ABB RobotStudio station: Project1.rsstnx

Station Project1 (saved by RobotStudio 24.3.10958.1)
Controller Controller1, task T_ROB1: task frame (RAPID world) sits at (0, 0, 500) mm in the station
Controller Controller1
  mechanical unit ROB_1: IRB660_180_315__01, 6 joints, base frame (0, 0, 0) mm
Layout (positions relative to the parent item):
  - IRB660_180_315__01 [mechanism, from %ABB.RobotStudio.Models.IRB660%\IRB660_180_315__01.rslib] at (0, 0, 500) mm; joint values [-0.0436, 0.6621, 0.6612, -0.0431] (rad or m)
  - SC_PM_PLC [smart component, from Components\SC_PM_PLC.rslib]
      properties: SimulationQuickStart=All; StatisticsInfo=; con0_ID={00f7108f-041a-4658-8432-4663a157ed6e}; con0_pmPLC_dpSelectedFlowID=7507beaf-a637-4325-82e6-8dabecadb5e7; con0_T_ROB1_ID={ede59ae2-37f1-49be-aecb-80bcdd7f86de}; con0_T_ROB1_ObjectReleased=(none); pf1_Product_ToPick={da9875e8-a75e-44a1-b53a-961bb916f098}; pf1_PreparationTime_ToPick=1; pf1_Product_Placed=; pf1_ClearTime_Placed=0; pf1_ID=4b299c2b-0326-42f9-880b-26203f6d833c; pf2_Product_ToPick=; pf2_PreparationTime_ToPick=0; pf2_Product_Placed={660944ae-43fb-4d62-84a1-2b4997365d4d}; pf2_ClearTime_Placed=1; pf2_ID=081b0045-7d90-402c-a41a-05ee4f4aed6a; pf3_Product_ToPick={55fdd2c5-2514-4d7a-936c-0e237c314134}; pf3_PreparationTime_ToPick=1; pf3_Product_Placed=; pf3_ClearTime_Placed=0; pf3_ID=f450dbdc-584e-4e57-b0ab-3fff9d44f94b
  - Part_1 [part] at (-700, -600, 0) mm, size 1200 x 1200 x 500 mm
  - FlexGripper 2.0_Vacuum_Pallet [smart component, from Grippers\FlexGripper 2.0_Vacuum_Pallet.rslib] at (2410.12, -105.03, 1233.55) mm, rotated rx 180 ry 0 rz 179.98 deg
      properties: ReleasedObject=(none)
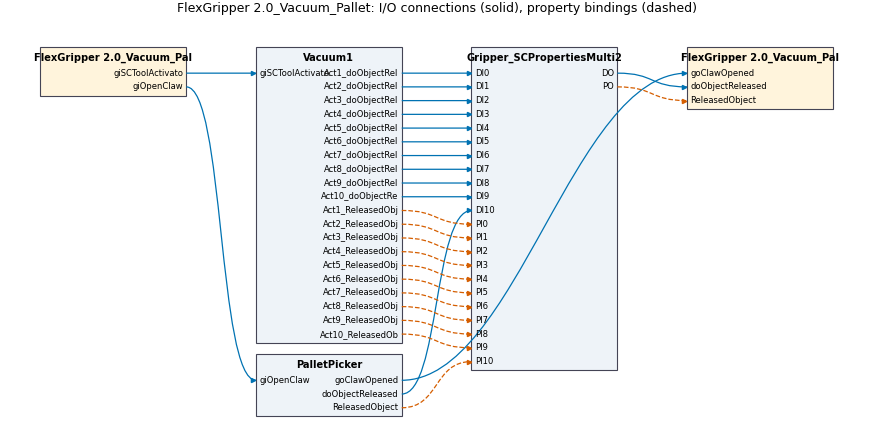
      connections:
        FlexGripper 2.0_Vacuum_Pallet.giSCToolActivators -> Vacuum1.giSCToolActivators
        FlexGripper 2.0_Vacuum_Pallet.giOpenClaw -> PalletPicker.giOpenClaw
        PalletPicker.goClawOpened -> FlexGripper 2.0_Vacuum_Pallet.goClawOpened
        Vacuum1.Act1_doObjectReleased -> Gripper_SCPropertiesMulti2Single.DI0
        Vacuum1.Act2_doObjectReleased -> Gripper_SCPropertiesMulti2Single.DI1
        Vacuum1.Act3_doObjectReleased -> Gripper_SCPropertiesMulti2Single.DI2
        Vacuum1.Act4_doObjectReleased -> Gripper_SCPropertiesMulti2Single.DI3
        Vacuum1.Act5_doObjectReleased -> Gripper_SCPropertiesMulti2Single.DI4
        Vacuum1.Act6_doObjectReleased -> Gripper_SCPropertiesMulti2Single.DI5
        Vacuum1.Act7_doObjectReleased -> Gripper_SCPropertiesMulti2Single.DI6
        Vacuum1.Act8_doObjectReleased -> Gripper_SCPropertiesMulti2Single.DI7
        Vacuum1.Act9_doObjectReleased -> Gripper_SCPropertiesMulti2Single.DI8
        Vacuum1.Act10_doObjectReleased -> Gripper_SCPropertiesMulti2Single.DI9
        PalletPicker.doObjectReleased -> Gripper_SCPropertiesMulti2Single.DI10
        Gripper_SCPropertiesMulti2Single.DO -> FlexGripper 2.0_Vacuum_Pallet.doObjectReleased
        Vacuum1.Act1_ReleasedObject => Gripper_SCPropertiesMulti2Single.PI0
        Vacuum1.Act2_ReleasedObject => Gripper_SCPropertiesMulti2Single.PI1
        Vacuum1.Act3_ReleasedObject => Gripper_SCPropertiesMulti2Single.PI2
        Vacuum1.Act4_ReleasedObject => Gripper_SCPropertiesMulti2Single.PI3
        Vacuum1.Act5_ReleasedObject => Gripper_SCPropertiesMulti2Single.PI4
        Vacuum1.Act6_ReleasedObject => Gripper_SCPropertiesMulti2Single.PI5
        Vacuum1.Act7_ReleasedObject => Gripper_SCPropertiesMulti2Single.PI6
        Vacuum1.Act8_ReleasedObject => Gripper_SCPropertiesMulti2Single.PI7
        Vacuum1.Act9_ReleasedObject => Gripper_SCPropertiesMulti2Single.PI8
        Vacuum1.Act10_ReleasedObject => Gripper_SCPropertiesMulti2Single.PI9
        PalletPicker.ReleasedObject => Gripper_SCPropertiesMulti2Single.PI10
        Gripper_SCPropertiesMulti2Single.PO => FlexGripper 2.0_Vacuum_Pallet.ReleasedObject
    - FlexGripper 2.0_Vacuum_Pallet [mechanism] at (0, 0, 0) mm; joint values [0, 0] (rad or m)
        TCP tVacuum at (0.12, 0.03, 163.81) mm, rotated rx 0 ry 0 rz -0.02 deg
        TCP tPalletPicker at (0.12, 0.03, 230.11) mm, rotated rx 0 ry 0 rz -0.02 deg
        links: L1, L2, L3, L4, L5, L6, L7
    - Vacuum1 [smart component]
        properties: Act1_ReleasedObject=(none); Act2_ReleasedObject=(none); Act3_ReleasedObject=(none); Act4_ReleasedObject=(none); Act5_ReleasedObject=(none); Act6_ReleasedObject=(none); Act7_ReleasedObject=(none); Act8_ReleasedObject=(none); Act9_ReleasedObject=(none); Act10_ReleasedObject=(none)
        signals: DO Act1_doObjectReleased, DO Act2_doObjectReleased, DO Act3_doObjectReleased, DO Act4_doObjectReleased, DO Act5_doObjectReleased, DO Act6_doObjectReleased, DO Act7_doObjectReleased, DO Act8_doObjectReleased, DO Act9_doObjectReleased, DO Act10_doObjectReleased, GI giSCToolActivators
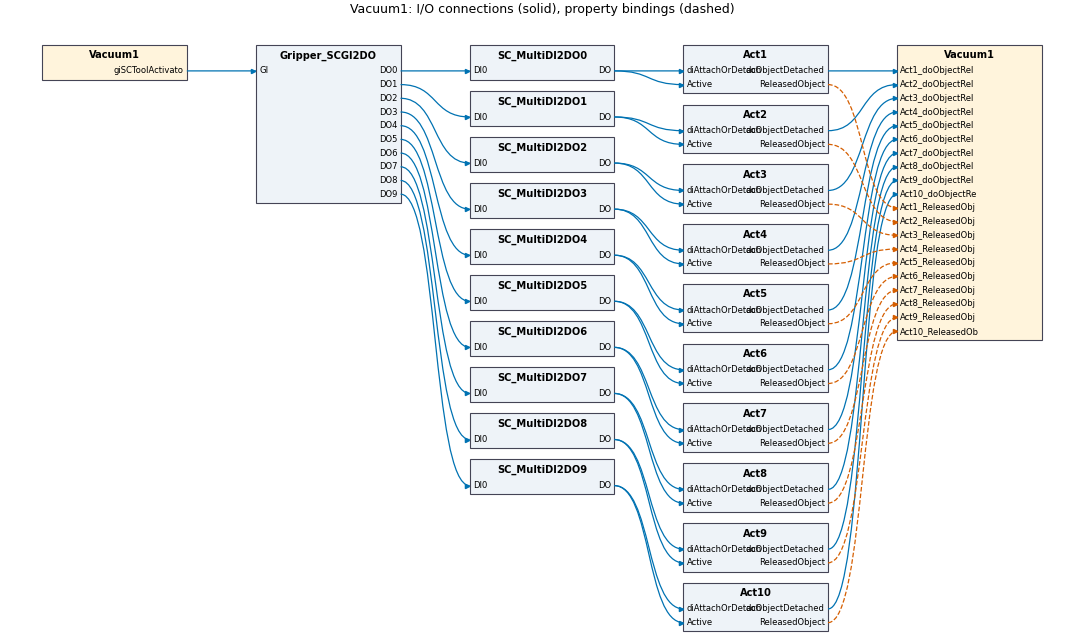
        connections:
          Act1.doObjectDetached -> Vacuum1.Act1_doObjectReleased
          Act2.doObjectDetached -> Vacuum1.Act2_doObjectReleased
          Act3.doObjectDetached -> Vacuum1.Act3_doObjectReleased
          Act4.doObjectDetached -> Vacuum1.Act4_doObjectReleased
          Act5.doObjectDetached -> Vacuum1.Act5_doObjectReleased
          Act6.doObjectDetached -> Vacuum1.Act6_doObjectReleased
          Act7.doObjectDetached -> Vacuum1.Act7_doObjectReleased
          Act8.doObjectDetached -> Vacuum1.Act8_doObjectReleased
          Act9.doObjectDetached -> Vacuum1.Act9_doObjectReleased
          Act10.doObjectDetached -> Vacuum1.Act10_doObjectReleased
          Gripper_SCGI2DO.DO0 -> SC_MultiDI2DO0.DI0
          SC_MultiDI2DO0.DO -> Act1.diAttachOrDetach
          SC_MultiDI2DO0.DO -> Act1.Active
          Gripper_SCGI2DO.DO1 -> SC_MultiDI2DO1.DI0
          SC_MultiDI2DO1.DO -> Act2.diAttachOrDetach
          SC_MultiDI2DO1.DO -> Act2.Active
          Gripper_SCGI2DO.DO2 -> SC_MultiDI2DO2.DI0
          SC_MultiDI2DO2.DO -> Act3.diAttachOrDetach
          SC_MultiDI2DO2.DO -> Act3.Active
          Gripper_SCGI2DO.DO3 -> SC_MultiDI2DO3.DI0
          SC_MultiDI2DO3.DO -> Act4.diAttachOrDetach
          SC_MultiDI2DO3.DO -> Act4.Active
          Gripper_SCGI2DO.DO4 -> SC_MultiDI2DO4.DI0
          SC_MultiDI2DO4.DO -> Act5.diAttachOrDetach
          SC_MultiDI2DO4.DO -> Act5.Active
          Gripper_SCGI2DO.DO5 -> SC_MultiDI2DO5.DI0
          SC_MultiDI2DO5.DO -> Act6.diAttachOrDetach
          SC_MultiDI2DO5.DO -> Act6.Active
          Gripper_SCGI2DO.DO6 -> SC_MultiDI2DO6.DI0
          SC_MultiDI2DO6.DO -> Act7.diAttachOrDetach
          SC_MultiDI2DO6.DO -> Act7.Active
          Gripper_SCGI2DO.DO7 -> SC_MultiDI2DO7.DI0
          SC_MultiDI2DO7.DO -> Act8.diAttachOrDetach
          SC_MultiDI2DO7.DO -> Act8.Active
          Gripper_SCGI2DO.DO8 -> SC_MultiDI2DO8.DI0
          SC_MultiDI2DO8.DO -> Act9.diAttachOrDetach
          SC_MultiDI2DO8.DO -> Act9.Active
          Gripper_SCGI2DO.DO9 -> SC_MultiDI2DO9.DI0
          SC_MultiDI2DO9.DO -> Act10.diAttachOrDetach
          SC_MultiDI2DO9.DO -> Act10.Active
          Vacuum1.giSCToolActivators -> Gripper_SCGI2DO.GI
          Act1.ReleasedObject => Vacuum1.Act1_ReleasedObject
          Act2.ReleasedObject => Vacuum1.Act2_ReleasedObject
          Act3.ReleasedObject => Vacuum1.Act3_ReleasedObject
          Act4.ReleasedObject => Vacuum1.Act4_ReleasedObject
          Act5.ReleasedObject => Vacuum1.Act5_ReleasedObject
          Act6.ReleasedObject => Vacuum1.Act6_ReleasedObject
          Act7.ReleasedObject => Vacuum1.Act7_ReleasedObject
          Act8.ReleasedObject => Vacuum1.Act8_ReleasedObject
          Act9.ReleasedObject => Vacuum1.Act9_ReleasedObject
          Act10.ReleasedObject => Vacuum1.Act10_ReleasedObject
      - Act1 [smart component] at (-0.1, -539.97, 163.81) mm, rotated rx 0 ry 0 rz -0.02 deg
          properties: ReleasedObject=(none); AttachedObject=(none)
          signals: DI diAttachOrDetach, DI Active, DO doObjectAttached, DO doObjectDetached
          connections:
            Act1.diAttachOrDetach -> SC_VolumeGripper.AttachOrDetach
            SC_VolumeGripper.TriggerAttach -> Attacher.Execute
            SC_VolumeGripper.TriggerDetach -> Detacher.Execute
            Attacher.Executed -> Act1.doObjectAttached
            Detacher.Executed -> Act1.doObjectDetached
            Act1.Active -> SC_VolumeGripper.Active
            SC_VolumeGripper.AttachParent => Attacher.Parent
            SC_VolumeGripper.ChildToAttach => Attacher.Child
            SC_VolumeGripper.AttachedChild => Detacher.Child
            SC_VolumeGripper.AttachedChild => Act1.AttachedObject
            SC_VolumeGripper.ReleasedChild => Act1.ReleasedObject
        - SC_VolumeGripper [smart component, from Components\SC_VolumeGripper.rslib]
            properties: Position=[0 0 0]; Orientation=[0 0 0]; Size=[0.28 0.1 0.02]; AttachParent=Act1; ChildToAttach=(none); AttachedChild=(none); ReleasedChild=(none)
          - _sensorPart_ [part], size 280 x 100 x 20 mm
        - Attacher [smart component, from Components\Attacher.rslib]
            properties: Parent=Act1; Flange=0; Child=(none); Mount=false; Offset=[0 0 0]; Orientation=[0 0 0]
        - Detacher [smart component, from Components\Detacher.rslib]
            properties: Child=(none); KeepPosition=true
      - Act2 [smart component] at (-0.05, -419.97, 163.81) mm, rotated rx 0 ry 0 rz -0.02 deg
          properties: ReleasedObject=(none); AttachedObject=(none)
          signals: DI diAttachOrDetach, DI Active, DO doObjectAttached, DO doObjectDetached
          connections:
            Act2.diAttachOrDetach -> SC_VolumeGripper.AttachOrDetach
            SC_VolumeGripper.TriggerAttach -> Attacher.Execute
            SC_VolumeGripper.TriggerDetach -> Detacher.Execute
            Attacher.Executed -> Act2.doObjectAttached
            Detacher.Executed -> Act2.doObjectDetached
            Act2.Active -> SC_VolumeGripper.Active
            SC_VolumeGripper.AttachParent => Attacher.Parent
            SC_VolumeGripper.ChildToAttach => Attacher.Child
            SC_VolumeGripper.AttachedChild => Detacher.Child
            SC_VolumeGripper.AttachedChild => Act2.AttachedObject
            SC_VolumeGripper.ReleasedChild => Act2.ReleasedObject
        - SC_VolumeGripper [smart component, from Components\SC_VolumeGripper.rslib]
            properties: Position=[0 0 0]; Orientation=[0 0 0]; Size=[0.28 0.1 0.02]; AttachParent=Act2; ChildToAttach=(none); AttachedChild=(none); ReleasedChild=(none)
          - _sensorPart_ [part], size 280 x 100 x 20 mm
        - Attacher [smart component, from Components\Attacher.rslib]
            properties: Parent=Act2; Flange=0; Child=(none); Mount=false; Offset=[0 0 0]; Orientation=[0 0 0]
        - Detacher [smart component, from Components\Detacher.rslib]
            properties: Child=(none); KeepPosition=true
      - Act3 [smart component] at (0, -299.97, 163.81) mm, rotated rx 0 ry 0 rz -0.02 deg
          properties: ReleasedObject=(none); AttachedObject=(none)
          signals: DI diAttachOrDetach, DI Active, DO doObjectAttached, DO doObjectDetached
          connections:
            Act3.diAttachOrDetach -> SC_VolumeGripper.AttachOrDetach
            SC_VolumeGripper.TriggerAttach -> Attacher.Execute
            SC_VolumeGripper.TriggerDetach -> Detacher.Execute
            Attacher.Executed -> Act3.doObjectAttached
            Detacher.Executed -> Act3.doObjectDetached
            Act3.Active -> SC_VolumeGripper.Active
            SC_VolumeGripper.AttachParent => Attacher.Parent
            SC_VolumeGripper.ChildToAttach => Attacher.Child
            SC_VolumeGripper.AttachedChild => Detacher.Child
            SC_VolumeGripper.AttachedChild => Act3.AttachedObject
            SC_VolumeGripper.ReleasedChild => Act3.ReleasedObject
        - SC_VolumeGripper [smart component, from Components\SC_VolumeGripper.rslib]
            properties: Position=[0 0 0]; Orientation=[0 0 0]; Size=[0.28 0.1 0.02]; AttachParent=Act3; ChildToAttach=(none); AttachedChild=(none); ReleasedChild=(none)
          - _sensorPart_ [part], size 280 x 100 x 20 mm
        - Attacher [smart component, from Components\Attacher.rslib]
            properties: Parent=Act3; Flange=0; Child=(none); Mount=false; Offset=[0 0 0]; Orientation=[0 0 0]
        - Detacher [smart component, from Components\Detacher.rslib]
            properties: Child=(none); KeepPosition=true
      - Act4 [smart component] at (0.05, -179.97, 163.81) mm, rotated rx 0 ry 0 rz -0.02 deg
          properties: ReleasedObject=(none); AttachedObject=(none)
          signals: DI diAttachOrDetach, DI Active, DO doObjectAttached, DO doObjectDetached
          connections:
            Act4.diAttachOrDetach -> SC_VolumeGripper.AttachOrDetach
            SC_VolumeGripper.TriggerAttach -> Attacher.Execute
            SC_VolumeGripper.TriggerDetach -> Detacher.Execute
            Attacher.Executed -> Act4.doObjectAttached
            Detacher.Executed -> Act4.doObjectDetached
            Act4.Active -> SC_VolumeGripper.Active
            SC_VolumeGripper.AttachParent => Attacher.Parent
            SC_VolumeGripper.ChildToAttach => Attacher.Child
            SC_VolumeGripper.AttachedChild => Detacher.Child
            SC_VolumeGripper.AttachedChild => Act4.AttachedObject
            SC_VolumeGripper.ReleasedChild => Act4.ReleasedObject
        - SC_VolumeGripper [smart component, from Components\SC_VolumeGripper.rslib]
            properties: Position=[0 0 0]; Orientation=[0 0 0]; Size=[0.28 0.1 0.02]; AttachParent=Act4; ChildToAttach=(none); AttachedChild=(none); ReleasedChild=(none)
          - _sensorPart_ [part], size 280 x 100 x 20 mm
        - Attacher [smart component, from Components\Attacher.rslib]
            properties: Parent=Act4; Flange=0; Child=(none); Mount=false; Offset=[0 0 0]; Orientation=[0 0 0]
        - Detacher [smart component, from Components\Detacher.rslib]
            properties: Child=(none); KeepPosition=true
      - Act5 [smart component] at (0.1, -59.97, 163.81) mm, rotated rx 0 ry 0 rz -0.02 deg
          properties: ReleasedObject=(none); AttachedObject=(none)
          signals: DI diAttachOrDetach, DI Active, DO doObjectAttached, DO doObjectDetached
          connections:
            Act5.diAttachOrDetach -> SC_VolumeGripper.AttachOrDetach
            SC_VolumeGripper.TriggerAttach -> Attacher.Execute
            SC_VolumeGripper.TriggerDetach -> Detacher.Execute
            Attacher.Executed -> Act5.doObjectAttached
            Detacher.Executed -> Act5.doObjectDetached
            Act5.Active -> SC_VolumeGripper.Active
            SC_VolumeGripper.AttachParent => Attacher.Parent
            SC_VolumeGripper.ChildToAttach => Attacher.Child
            SC_VolumeGripper.AttachedChild => Detacher.Child
            SC_VolumeGripper.AttachedChild => Act5.AttachedObject
            SC_VolumeGripper.ReleasedChild => Act5.ReleasedObject
        - SC_VolumeGripper [smart component, from Components\SC_VolumeGripper.rslib]
            properties: Position=[0 0 0]; Orientation=[0 0 0]; Size=[0.28 0.1 0.02]; AttachParent=Act5; ChildToAttach=(none); AttachedChild=(none); ReleasedChild=(none)
          - _sensorPart_ [part], size 280 x 100 x 20 mm
        - Attacher [smart component, from Components\Attacher.rslib]
            properties: Parent=Act5; Flange=0; Child=(none); Mount=false; Offset=[0 0 0]; Orientation=[0 0 0]
        - Detacher [smart component, from Components\Detacher.rslib]
            properties: Child=(none); KeepPosition=true
      - Act6 [smart component] at (0.14, 60.03, 163.81) mm, rotated rx 0 ry 0 rz -0.02 deg
          properties: ReleasedObject=(none); AttachedObject=(none)
          signals: DI diAttachOrDetach, DI Active, DO doObjectAttached, DO doObjectDetached
          connections:
            Act6.diAttachOrDetach -> SC_VolumeGripper.AttachOrDetach
            SC_VolumeGripper.TriggerAttach -> Attacher.Execute
            SC_VolumeGripper.TriggerDetach -> Detacher.Execute
            Attacher.Executed -> Act6.doObjectAttached
            Detacher.Executed -> Act6.doObjectDetached
            Act6.Active -> SC_VolumeGripper.Active
            SC_VolumeGripper.AttachParent => Attacher.Parent
            SC_VolumeGripper.ChildToAttach => Attacher.Child
            SC_VolumeGripper.AttachedChild => Detacher.Child
            SC_VolumeGripper.AttachedChild => Act6.AttachedObject
            SC_VolumeGripper.ReleasedChild => Act6.ReleasedObject
        - SC_VolumeGripper [smart component, from Components\SC_VolumeGripper.rslib]
            properties: Position=[0 0 0]; Orientation=[0 0 0]; Size=[0.28 0.1 0.02]; AttachParent=Act6; ChildToAttach=(none); AttachedChild=(none); ReleasedChild=(none)
          - _sensorPart_ [part], size 280 x 100 x 20 mm
        - Attacher [smart component, from Components\Attacher.rslib]
            properties: Parent=Act6; Flange=0; Child=(none); Mount=false; Offset=[0 0 0]; Orientation=[0 0 0]
        - Detacher [smart component, from Components\Detacher.rslib]
            properties: Child=(none); KeepPosition=true
      - Act7 [smart component] at (0.19, 180.03, 163.81) mm, rotated rx 0 ry 0 rz -0.02 deg
          properties: ReleasedObject=(none); AttachedObject=(none)
          signals: DI diAttachOrDetach, DI Active, DO doObjectAttached, DO doObjectDetached
          connections:
            Act7.diAttachOrDetach -> SC_VolumeGripper.AttachOrDetach
            SC_VolumeGripper.TriggerAttach -> Attacher.Execute
            SC_VolumeGripper.TriggerDetach -> Detacher.Execute
            Attacher.Executed -> Act7.doObjectAttached
            Detacher.Executed -> Act7.doObjectDetached
            Act7.Active -> SC_VolumeGripper.Active
            SC_VolumeGripper.AttachParent => Attacher.Parent
            SC_VolumeGripper.ChildToAttach => Attacher.Child
            SC_VolumeGripper.AttachedChild => Detacher.Child
            SC_VolumeGripper.AttachedChild => Act7.AttachedObject
            SC_VolumeGripper.ReleasedChild => Act7.ReleasedObject
        - SC_VolumeGripper [smart component, from Components\SC_VolumeGripper.rslib]
            properties: Position=[0 0 0]; Orientation=[0 0 0]; Size=[0.28 0.1 0.02]; AttachParent=Act7; ChildToAttach=(none); AttachedChild=(none); ReleasedChild=(none)
          - _sensorPart_ [part], size 280 x 100 x 20 mm
        - Attacher [smart component, from Components\Attacher.rslib]
            properties: Parent=Act7; Flange=0; Child=(none); Mount=false; Offset=[0 0 0]; Orientation=[0 0 0]
        - Detacher [smart component, from Components\Detacher.rslib]
            properties: Child=(none); KeepPosition=true
      - Act8 [smart component] at (0.24, 300.03, 163.81) mm, rotated rx 0 ry 0 rz -0.02 deg
          properties: ReleasedObject=(none); AttachedObject=(none)
          signals: DI diAttachOrDetach, DI Active, DO doObjectAttached, DO doObjectDetached
          connections:
            Act8.diAttachOrDetach -> SC_VolumeGripper.AttachOrDetach
            SC_VolumeGripper.TriggerAttach -> Attacher.Execute
            SC_VolumeGripper.TriggerDetach -> Detacher.Execute
            Attacher.Executed -> Act8.doObjectAttached
            Detacher.Executed -> Act8.doObjectDetached
            Act8.Active -> SC_VolumeGripper.Active
            SC_VolumeGripper.AttachParent => Attacher.Parent
            SC_VolumeGripper.ChildToAttach => Attacher.Child
            SC_VolumeGripper.AttachedChild => Detacher.Child
            SC_VolumeGripper.AttachedChild => Act8.AttachedObject
            SC_VolumeGripper.ReleasedChild => Act8.ReleasedObject
        - SC_VolumeGripper [smart component, from Components\SC_VolumeGripper.rslib]
            properties: Position=[0 0 0]; Orientation=[0 0 0]; Size=[0.28 0.1 0.02]; AttachParent=Act8; ChildToAttach=(none); AttachedChild=(none); ReleasedChild=(none)
          - _sensorPart_ [part], size 280 x 100 x 20 mm
        - Attacher [smart component, from Components\Attacher.rslib]
            properties: Parent=Act8; Flange=0; Child=(none); Mount=false; Offset=[0 0 0]; Orientation=[0 0 0]
        - Detacher [smart component, from Components\Detacher.rslib]
            properties: Child=(none); KeepPosition=true
      - Act9 [smart component] at (0.29, 420.03, 163.81) mm, rotated rx 0 ry 0 rz -0.02 deg
          properties: ReleasedObject=(none); AttachedObject=(none)
          signals: DI diAttachOrDetach, DI Active, DO doObjectAttached, DO doObjectDetached
          connections:
            Act9.diAttachOrDetach -> SC_VolumeGripper.AttachOrDetach
            SC_VolumeGripper.TriggerAttach -> Attacher.Execute
            SC_VolumeGripper.TriggerDetach -> Detacher.Execute
            Attacher.Executed -> Act9.doObjectAttached
            Detacher.Executed -> Act9.doObjectDetached
            Act9.Active -> SC_VolumeGripper.Active
            SC_VolumeGripper.AttachParent => Attacher.Parent
            SC_VolumeGripper.ChildToAttach => Attacher.Child
            SC_VolumeGripper.AttachedChild => Detacher.Child
            SC_VolumeGripper.AttachedChild => Act9.AttachedObject
            SC_VolumeGripper.ReleasedChild => Act9.ReleasedObject
        - SC_VolumeGripper [smart component, from Components\SC_VolumeGripper.rslib]
            properties: Position=[0 0 0]; Orientation=[0 0 0]; Size=[0.28 0.1 0.02]; AttachParent=Act9; ChildToAttach=(none); AttachedChild=(none); ReleasedChild=(none)
          - _sensorPart_ [part], size 280 x 100 x 20 mm
        - Attacher [smart component, from Components\Attacher.rslib]
            properties: Parent=Act9; Flange=0; Child=(none); Mount=false; Offset=[0 0 0]; Orientation=[0 0 0]
        - Detacher [smart component, from Components\Detacher.rslib]
            properties: Child=(none); KeepPosition=true
      - Act10 [smart component] at (0.34, 540.03, 163.81) mm, rotated rx 0 ry 0 rz -0.02 deg
          properties: ReleasedObject=(none); AttachedObject=(none)
          signals: DI diAttachOrDetach, DI Active, DO doObjectAttached, DO doObjectDetached
          connections:
            Act10.diAttachOrDetach -> SC_VolumeGripper.AttachOrDetach
            SC_VolumeGripper.TriggerAttach -> Attacher.Execute
            SC_VolumeGripper.TriggerDetach -> Detacher.Execute
            Attacher.Executed -> Act10.doObjectAttached
            Detacher.Executed -> Act10.doObjectDetached
            Act10.Active -> SC_VolumeGripper.Active
            SC_VolumeGripper.AttachParent => Attacher.Parent
            SC_VolumeGripper.ChildToAttach => Attacher.Child
            SC_VolumeGripper.AttachedChild => Detacher.Child
            SC_VolumeGripper.AttachedChild => Act10.AttachedObject
            SC_VolumeGripper.ReleasedChild => Act10.ReleasedObject
        - SC_VolumeGripper [smart component, from Components\SC_VolumeGripper.rslib]
            properties: Position=[0 0 0]; Orientation=[0 0 0]; Size=[0.28 0.1 0.02]; AttachParent=Act10; ChildToAttach=(none); AttachedChild=(none); ReleasedChild=(none)
          - _sensorPart_ [part], size 280 x 100 x 20 mm
        - Attacher [smart component, from Components\Attacher.rslib]
            properties: Parent=Act10; Flange=0; Child=(none); Mount=false; Offset=[0 0 0]; Orientation=[0 0 0]
        - Detacher [smart component, from Components\Detacher.rslib]
            properties: Child=(none); KeepPosition=true
      - Gripper_SCGI2DO [smart component, from Components\SC_GI2DO.rslib]
          properties: DOCount=11
      - SC_MultiDI2DO0 [smart component, from Components\SC_MultiDI2DO.rslib]
          properties: DICount=1; ConnectionType=0/1
      - SC_MultiDI2DO1 [smart component, from Components\SC_MultiDI2DO.rslib]
          properties: DICount=1; ConnectionType=0/1
      - SC_MultiDI2DO2 [smart component, from Components\SC_MultiDI2DO.rslib]
          properties: DICount=1; ConnectionType=0/1
      - SC_MultiDI2DO3 [smart component, from Components\SC_MultiDI2DO.rslib]
          properties: DICount=1; ConnectionType=0/1
      - SC_MultiDI2DO4 [smart component, from Components\SC_MultiDI2DO.rslib]
          properties: DICount=1; ConnectionType=0/1
      - SC_MultiDI2DO5 [smart component, from Components\SC_MultiDI2DO.rslib]
          properties: DICount=1; ConnectionType=0/1
      - SC_MultiDI2DO6 [smart component, from Components\SC_MultiDI2DO.rslib]
          properties: DICount=1; ConnectionType=0/1
      - SC_MultiDI2DO7 [smart component, from Components\SC_MultiDI2DO.rslib]
          properties: DICount=1; ConnectionType=0/1
      - SC_MultiDI2DO8 [smart component, from Components\SC_MultiDI2DO.rslib]
          properties: DICount=1; ConnectionType=0/1
      - SC_MultiDI2DO9 [smart component, from Components\SC_MultiDI2DO.rslib]
          properties: DICount=1; ConnectionType=0/1
    - PalletPicker [smart component]
        properties: ReleasedObject=(none)
        signals: GI giOpenClaw, GO goClawOpened, DO doObjectReleased
        connections:
          PalletPicker.giOpenClaw -> ClawControl.giOpenClaw
          ClawControl.goClawOpened -> PalletPicker.goClawOpened
          ClawAct.doObjectDetached -> PalletPicker.doObjectReleased
          ClawControl.Closed -> LogicSRLatch.Set
          ClawControl.Opening -> LogicSRLatch.Reset
          LogicSRLatch.Output -> ClawAct.diAttachOrDetach
          ClawControl.Closed -> LogicGate.InputA
          ClawControl.Opening -> LogicGate.InputB
          LogicGate.Output -> ClawAct.Active
          ClawAct.ReleasedObject => PalletPicker.ReleasedObject
      - ClawControl [smart component]
          signals: GI giOpenClaw, GO goClawOpened, DO Closing, DO Closed, DO Opening, DO Opened
          connections:
            JointMoverClose.Executing -> ClawControl.Closing
            JointMoverClose.Executed -> ClawControl.Closed
            JointMoverOpen.Executing -> ClawControl.Opening
            JointMoverOpen.Executed -> ClawControl.Opened
            ClawControl.giOpenClaw -> MultiSignalJudgeOpen.GI0
            MultiSignalJudgeOpen.DO -> JointMoverOpen.Execute
            JointMoverOpen.Executed -> MultiSignalSetOpen.Set
            ClawControl.giOpenClaw -> MultiSignalJudgeClose.GI0
            MultiSignalJudgeClose.DO -> JointMoverClose.Execute
            JointMoverClose.Executed -> MultiSignalSetClose.Set
            MultiSignalSetOpen.Executed -> MutiSignalSelector.SelectorA
            MultiSignalSetOpen.GO0 -> MutiSignalSelector.GiA0
            MultiSignalSetClose.Executed -> MutiSignalSelector.SelectorB
            MultiSignalSetClose.GO0 -> MutiSignalSelector.GiB0
            MutiSignalSelector.goClawOpened -> ClawControl.goClawOpened
        - MultiSignalJudgeOpen [smart component, from Components\SC_MultiSignalJudge.rslib]
            properties: DICount=0; GICount=1
        - JointMoverOpen [smart component, from Components\SC_JointMoverEx.rslib]
            properties: Mechanism=FlexGripper 2.0_Vacuum_Pallet; Relative=false; Duration=0.5; UseJ1=true; J1=0.1; UseJ2=true; J2=0.1
        - MultiSignalSetOpen [smart component, from Components\SC_MultiSignalSet.rslib]
            properties: DOCount=0; GOCount=1
        - MultiSignalJudgeClose [smart component, from Components\SC_MultiSignalJudge.rslib]
            properties: DICount=0; GICount=1
        - JointMoverClose [smart component, from Components\SC_JointMoverEx.rslib]
            properties: Mechanism=FlexGripper 2.0_Vacuum_Pallet; Relative=false; Duration=0.5; UseJ1=true; J1=0; UseJ2=true; J2=0
        - MultiSignalSetClose [smart component, from Components\SC_MultiSignalSet.rslib]
            properties: DOCount=0; GOCount=1
        - MutiSignalSelector [smart component, from Components\SC_MultiSignalSelector.rslib]
            properties: DICountA=0; GICountA=1; DICountB=0; GICountB=1; PiGiA0=goClawOpened; PiGiB0=goClawOpened
      - ClawAct [smart component] at (0.12, 0.03, 180.11) mm, rotated rx 0 ry 0 rz -0.02 deg
          properties: ReleasedObject=(none); AttachedObject=(none)
          signals: DI diAttachOrDetach, DI Active, DO doObjectAttached, DO doObjectDetached
          connections:
            ClawAct.diAttachOrDetach -> SC_VolumeGripper.AttachOrDetach
            SC_VolumeGripper.TriggerAttach -> Attacher.Execute
            SC_VolumeGripper.TriggerDetach -> Detacher.Execute
            Attacher.Executed -> ClawAct.doObjectAttached
            Detacher.Executed -> ClawAct.doObjectDetached
            ClawAct.Active -> SC_VolumeGripper.Active
            SC_VolumeGripper.AttachParent => Attacher.Parent
            SC_VolumeGripper.ChildToAttach => Attacher.Child
            SC_VolumeGripper.AttachedChild => Detacher.Child
            SC_VolumeGripper.AttachedChild => ClawAct.AttachedObject
            SC_VolumeGripper.ReleasedChild => ClawAct.ReleasedObject
        - SC_VolumeGripper [smart component, from Components\SC_VolumeGripper.rslib]
            properties: Position=[0 0 0]; Orientation=[0 0 0]; Size=[0.02 1.2 0.08]; AttachParent=ClawAct; ChildToAttach=(none); AttachedChild=(none); ReleasedChild=(none)
          - _sensorPart_ [part], size 20 x 1200 x 80 mm
        - Attacher [smart component, from Components\Attacher.rslib]
            properties: Parent=ClawAct; Flange=0; Child=(none); Mount=false; Offset=[0 0 0]; Orientation=[0 0 0]
        - Detacher [smart component, from Components\Detacher.rslib]
            properties: Child=(none); KeepPosition=true
      - LogicSRLatch [smart component, from Components\LogicSRLatch.rslib]
      - LogicGate [smart component, from Components\LogicGate.rslib]
          properties: Operator=OR; Delay=0
    - Gripper_SCPropertiesMulti2Single [smart component, from Components\SC_PropertiesMulti2Single.rslib]
        properties: Count=11; PO=(none); PI0=(none); PI1=(none); PI2=(none); PI3=(none); PI4=(none); PI5=(none); PI6=(none); PI7=(none); PI8=(none); PI9=(none); PI10=(none)
  - Conveyor_600 [smart component, from Feeders\Conveyor_600.rslib] at (800, 2100, 0) mm, rotated rx 0 ry 0 rz 90 deg
      properties: PreparationTime_ToPick=1; Product_ToPick={da9875e8-a75e-44a1-b53a-961bb916f098}; ClearTime_Placed=0; Product_Placed=
      connections:
        Conveyor_600.Reset -> SCFeederController.Reset
        Conveyor_600.Enqueue_ToPick -> SCFeederController.Enqueue_ToPick
        SCFeederController.Shown_ToPick -> Conveyor_600.Shown_ToPick
        Conveyor_600.Clear_ToPick -> SCFeederController.Clear_ToPick
        Conveyor_600.GI_ProdSel_ToPick -> SCFeederController.GI_ProdSel_ToPick
        Conveyor_600.GI_FormSel_ToPick -> SCFeederController.GI_FormSel_ToPick
        SCFeederController.GO_ProdSel_ToPick -> Conveyor_600.GO_ProdSel_ToPick
        SCFeederController.GO_FormSel_ToPick -> Conveyor_600.GO_FormSel_ToPick
        SCFeederController.Clear_Placed_Finished -> Conveyor_600.Clear_Placed_Finished
        Conveyor_600.Enqueue_Placed -> SCFeederController.Enqueue_Placed
        Conveyor_600.Clear_Placed -> SCFeederController.Clear_Placed
        Conveyor_600.Enqueue_IOPlacedRequest -> SCFeederController.Enqueue_IOPlacedRequest
        Conveyor_600.GI_ProdSel_PlacedRequest -> SCFeederController.GI_ProdSel_PlacedRequest
        Conveyor_600.GI_FormSel_PlacedRequest -> SCFeederController.GI_FormSel_PlacedRequest
        SCFeederController.GO_ProdSel_PlacedRequest -> Conveyor_600.GO_ProdSel_PlacedRequest
        SCFeederController.GO_FormSel_PlacedRequest -> Conveyor_600.GO_FormSel_PlacedRequest
        SCFeederController.IsReady_IOPlacedRequest -> Conveyor_600.IsReady_IOPlacedRequest
        Conveyor_600.PreparationTime_ToPick => SCFeederController.PreparationTime_ToPick
        Conveyor_600.Product_ToPick => SCFeederController.Product_ToPick
        Conveyor_600.ClearTime_Placed => SCFeederController.ClearTime_Placed
        Conveyor_600.Product_Placed => SCFeederController.Product_Placed
    - 600_guide [part, from Feeders\Conveyor_600.rslib]
    - SCFeederController [smart component, from Components\SC_FeederController.rslib]
        properties: Product_Placed=; ClearTime_Placed=0; PreparationTime_ToPick=1; Product_ToPick={da9875e8-a75e-44a1-b53a-961bb916f098}
  - Outfeeder_1320 [smart component, from Feeders\Outfeeder_1320.rslib] at (1600, -700, 0) mm
      properties: PreparationTime_ToPick=0; Product_ToPick=; ClearTime_Placed=1; Product_Placed={660944ae-43fb-4d62-84a1-2b4997365d4d}
      connections:
        Outfeeder_1320.Reset -> SCFeederController.Reset
        Outfeeder_1320.Enqueue_ToPick -> SCFeederController.Enqueue_ToPick
        SCFeederController.Shown_ToPick -> Outfeeder_1320.Shown_ToPick
        Outfeeder_1320.Clear_ToPick -> SCFeederController.Clear_ToPick
        Outfeeder_1320.GI_ProdSel_ToPick -> SCFeederController.GI_ProdSel_ToPick
        Outfeeder_1320.GI_FormSel_ToPick -> SCFeederController.GI_FormSel_ToPick
        SCFeederController.GO_ProdSel_ToPick -> Outfeeder_1320.GO_ProdSel_ToPick
        SCFeederController.GO_FormSel_ToPick -> Outfeeder_1320.GO_FormSel_ToPick
        SCFeederController.Clear_Placed_Finished -> Outfeeder_1320.Clear_Placed_Finished
        Outfeeder_1320.Enqueue_Placed -> SCFeederController.Enqueue_Placed
        Outfeeder_1320.Clear_Placed -> SCFeederController.Clear_Placed
        Outfeeder_1320.Enqueue_IOPlacedRequest -> SCFeederController.Enqueue_IOPlacedRequest
        Outfeeder_1320.GI_ProdSel_PlacedRequest -> SCFeederController.GI_ProdSel_PlacedRequest
        Outfeeder_1320.GI_FormSel_PlacedRequest -> SCFeederController.GI_FormSel_PlacedRequest
        SCFeederController.GO_ProdSel_PlacedRequest -> Outfeeder_1320.GO_ProdSel_PlacedRequest
        SCFeederController.GO_FormSel_PlacedRequest -> Outfeeder_1320.GO_FormSel_PlacedRequest
        SCFeederController.IsReady_IOPlacedRequest -> Outfeeder_1320.IsReady_IOPlacedRequest
        Outfeeder_1320.PreparationTime_ToPick => SCFeederController.PreparationTime_ToPick
        Outfeeder_1320.Product_ToPick => SCFeederController.Product_ToPick
        Outfeeder_1320.ClearTime_Placed => SCFeederController.ClearTime_Placed
        Outfeeder_1320.Product_Placed => SCFeederController.Product_Placed
    - 1320_4000_h2 [part, from Feeders\Outfeeder_1320.rslib]
    - SCFeederController [smart component, from Components\SC_FeederController.rslib]
        properties: Product_Placed={660944ae-43fb-4d62-84a1-2b4997365d4d}; ClearTime_Placed=1; PreparationTime_ToPick=0; Product_ToPick=
  - PalletDispenser 1300_1300_300 [smart component, from Feeders\PalletDispenser 1300_1300_300.rslib] at (-300, -1600, 0) mm, rotated rx 0 ry 0 rz -90 deg
      properties: PreparationTime_ToPick=1; Product_ToPick={55fdd2c5-2514-4d7a-936c-0e237c314134}; ClearTime_Placed=0; Product_Placed=
      connections:
        PalletDispenser 1300_1300_300.Reset -> SCFeederController.Reset
        PalletDispenser 1300_1300_300.Enqueue_ToPick -> SCFeederController.Enqueue_ToPick
        SCFeederController.Shown_ToPick -> PalletDispenser 1300_1300_300.Shown_ToPick
        PalletDispenser 1300_1300_300.Clear_ToPick -> SCFeederController.Clear_ToPick
        PalletDispenser 1300_1300_300.GI_ProdSel_ToPick -> SCFeederController.GI_ProdSel_ToPick
        PalletDispenser 1300_1300_300.GI_FormSel_ToPick -> SCFeederController.GI_FormSel_ToPick
        SCFeederController.GO_ProdSel_ToPick -> PalletDispenser 1300_1300_300.GO_ProdSel_ToPick
        SCFeederController.GO_FormSel_ToPick -> PalletDispenser 1300_1300_300.GO_FormSel_ToPick
        SCFeederController.Clear_Placed_Finished -> PalletDispenser 1300_1300_300.Clear_Placed_Finished
        PalletDispenser 1300_1300_300.Enqueue_Placed -> SCFeederController.Enqueue_Placed
        PalletDispenser 1300_1300_300.Clear_Placed -> SCFeederController.Clear_Placed
        PalletDispenser 1300_1300_300.Enqueue_IOPlacedRequest -> SCFeederController.Enqueue_IOPlacedRequest
        PalletDispenser 1300_1300_300.GI_ProdSel_PlacedRequest -> SCFeederController.GI_ProdSel_PlacedRequest
        PalletDispenser 1300_1300_300.GI_FormSel_PlacedRequest -> SCFeederController.GI_FormSel_PlacedRequest
        SCFeederController.GO_ProdSel_PlacedRequest -> PalletDispenser 1300_1300_300.GO_ProdSel_PlacedRequest
        SCFeederController.GO_FormSel_PlacedRequest -> PalletDispenser 1300_1300_300.GO_FormSel_PlacedRequest
        SCFeederController.IsReady_IOPlacedRequest -> PalletDispenser 1300_1300_300.IsReady_IOPlacedRequest
        PalletDispenser 1300_1300_300.PreparationTime_ToPick => SCFeederController.PreparationTime_ToPick
        PalletDispenser 1300_1300_300.Product_ToPick => SCFeederController.Product_ToPick
        PalletDispenser 1300_1300_300.ClearTime_Placed => SCFeederController.ClearTime_Placed
        PalletDispenser 1300_1300_300.Product_Placed => SCFeederController.Product_Placed
    - PalletDispenser 1300_1300_300 [part, from Feeders\PalletDispenser 1300_1300_300.rslib]
    - SCFeederController [smart component, from Components\SC_FeederController.rslib]
        properties: Product_Placed=; ClearTime_Placed=0; PreparationTime_ToPick=1; Product_ToPick={55fdd2c5-2514-4d7a-936c-0e237c314134}
  - PalletPattern1 [graphiccomponentgroup] at (1660, 580, 419.75) mm, rotated rx 0 ry 0 rz -90 deg
  - Box1 [graphiccomponentgroup] at (0, 0, -2201.5) mm
    - MainBody [part], size 500 x 300 x 200 mm
    - OuterLine [part], size 500 x 300 x 200 mm
    - Labels [part], size 150 x 150 x 0 mm
    - Origin [part], size 100.5 x 60.5 x 201 mm
  - Pallet1 [graphiccomponentgroup] at (0, 0, -2151.5) mm
    - MainBody [part], size 1200 x 1000 x 150 mm
    - OuterLine [part], size 1200 x 1000 x 150 mm
    - Labels [part], size 500 x 500 x 0 mm
    - Origin [part], size 240.5 x 200.5 x 151 mm
Attachment: FlexGripper 2.0_Vacuum_Pallet is attached to IRB660_180_315__01 / Link6
Attachment: pmInfeeder1_WObj is attached to Conveyor_600
Attachment: pmOutfeeder1_WObj is attached to Outfeeder_1320
Attachment: pmPallet1_WObj is attached to PalletDispenser 1300_1300_300
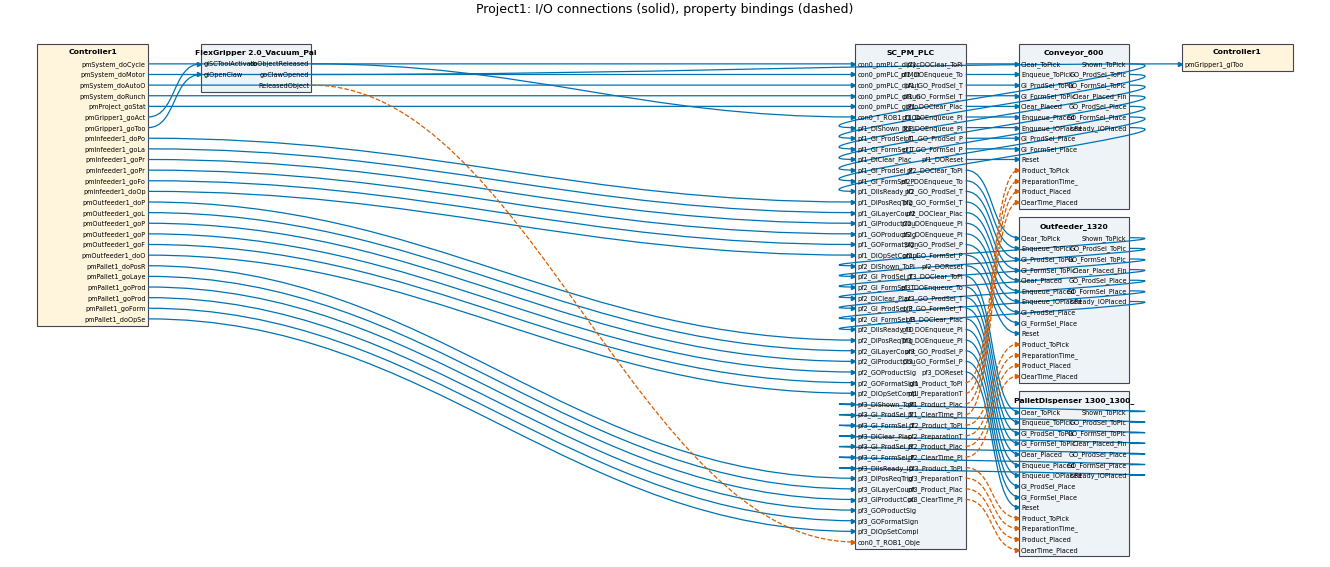
Station logic (signal -> signal, property => property):
  Controller1.pmSystem_doCycleOn -> SC_PM_PLC.con0_pmPLC_diCycleOn
  Controller1.pmSystem_doMotorOn -> SC_PM_PLC.con0_pmPLC_diMotorOn
  Controller1.pmSystem_doAutoOn -> SC_PM_PLC.con0_pmPLC_diAutoOn
  Controller1.pmSystem_doRunchOk -> SC_PM_PLC.con0_pmPLC_diRunchOk
  Controller1.pmProject_goStatus -> SC_PM_PLC.con0_pmPLC_giProjectStatus
  FlexGripper 2.0_Vacuum_Pallet.doObjectReleased -> SC_PM_PLC.con0_T_ROB1_DIObjectReleased
  Controller1.pmGripper1_goActivators -> FlexGripper 2.0_Vacuum_Pallet.giSCToolActivators
  Controller1.pmGripper1_goToolEvent1 -> FlexGripper 2.0_Vacuum_Pallet.giOpenClaw
  FlexGripper 2.0_Vacuum_Pallet.goClawOpened -> Controller1.pmGripper1_giToolEvent1
  Conveyor_600.Shown_ToPick -> SC_PM_PLC.pf1_DIShown_ToPick
  SC_PM_PLC.pf1_DOClear_ToPick -> Conveyor_600.Clear_ToPick
  SC_PM_PLC.pf1_DOEnqueue_ToPick -> Conveyor_600.Enqueue_ToPick
  Conveyor_600.GO_ProdSel_ToPick -> SC_PM_PLC.pf1_GI_ProdSel_ToPick
  Conveyor_600.GO_FormSel_ToPick -> SC_PM_PLC.pf1_GI_FormSel_ToPick
  SC_PM_PLC.pf1_GO_ProdSel_ToPick -> Conveyor_600.GI_ProdSel_ToPick
  SC_PM_PLC.pf1_GO_FormSel_ToPick -> Conveyor_600.GI_FormSel_ToPick
  Conveyor_600.Clear_Placed_Finished -> SC_PM_PLC.pf1_DIClear_Placed_Finished
  SC_PM_PLC.pf1_DOClear_Placed -> Conveyor_600.Clear_Placed
  SC_PM_PLC.pf1_DOEnqueue_Placed -> Conveyor_600.Enqueue_Placed
  SC_PM_PLC.pf1_DOEnqueue_PlacedRequest -> Conveyor_600.Enqueue_IOPlacedRequest
  Conveyor_600.GO_ProdSel_PlacedRequest -> SC_PM_PLC.pf1_GI_ProdSel_PlacedRequest
  Conveyor_600.GO_FormSel_PlacedRequest -> SC_PM_PLC.pf1_GI_FormSel_PlacedRequest
  SC_PM_PLC.pf1_GO_ProdSel_PlacedRequest -> Conveyor_600.GI_ProdSel_PlacedRequest
  SC_PM_PLC.pf1_GO_FormSel_PlacedRequest -> Conveyor_600.GI_FormSel_PlacedRequest
  Conveyor_600.IsReady_IOPlacedRequest -> SC_PM_PLC.pf1_DIIsReady_IOPlacedRequest
  SC_PM_PLC.pf1_DOReset -> Conveyor_600.Reset
  Controller1.pmInfeeder1_doPosReqTrig -> SC_PM_PLC.pf1_DIPosReqTrig
  Controller1.pmInfeeder1_goLayerCount -> SC_PM_PLC.pf1_GILayerCount
  Controller1.pmInfeeder1_goProductCount -> SC_PM_PLC.pf1_GIProductCount
  Controller1.pmInfeeder1_goProduct -> SC_PM_PLC.pf1_GOProductSignal
  Controller1.pmInfeeder1_goFormat -> SC_PM_PLC.pf1_GOFormatSignal
  Controller1.pmInfeeder1_doOpSetCompl -> SC_PM_PLC.pf1_DIOpSetCompl
  Outfeeder_1320.Shown_ToPick -> SC_PM_PLC.pf2_DIShown_ToPick
  SC_PM_PLC.pf2_DOClear_ToPick -> Outfeeder_1320.Clear_ToPick
  SC_PM_PLC.pf2_DOEnqueue_ToPick -> Outfeeder_1320.Enqueue_ToPick
  Outfeeder_1320.GO_ProdSel_ToPick -> SC_PM_PLC.pf2_GI_ProdSel_ToPick
  Outfeeder_1320.GO_FormSel_ToPick -> SC_PM_PLC.pf2_GI_FormSel_ToPick
  SC_PM_PLC.pf2_GO_ProdSel_ToPick -> Outfeeder_1320.GI_ProdSel_ToPick
  SC_PM_PLC.pf2_GO_FormSel_ToPick -> Outfeeder_1320.GI_FormSel_ToPick
  Outfeeder_1320.Clear_Placed_Finished -> SC_PM_PLC.pf2_DIClear_Placed_Finished
  SC_PM_PLC.pf2_DOClear_Placed -> Outfeeder_1320.Clear_Placed
  SC_PM_PLC.pf2_DOEnqueue_Placed -> Outfeeder_1320.Enqueue_Placed
  SC_PM_PLC.pf2_DOEnqueue_PlacedRequest -> Outfeeder_1320.Enqueue_IOPlacedRequest
  Outfeeder_1320.GO_ProdSel_PlacedRequest -> SC_PM_PLC.pf2_GI_ProdSel_PlacedRequest
  Outfeeder_1320.GO_FormSel_PlacedRequest -> SC_PM_PLC.pf2_GI_FormSel_PlacedRequest
  SC_PM_PLC.pf2_GO_ProdSel_PlacedRequest -> Outfeeder_1320.GI_ProdSel_PlacedRequest
  SC_PM_PLC.pf2_GO_FormSel_PlacedRequest -> Outfeeder_1320.GI_FormSel_PlacedRequest
  Outfeeder_1320.IsReady_IOPlacedRequest -> SC_PM_PLC.pf2_DIIsReady_IOPlacedRequest
  SC_PM_PLC.pf2_DOReset -> Outfeeder_1320.Reset
  Controller1.pmOutfeeder1_doPosReqTrig -> SC_PM_PLC.pf2_DIPosReqTrig
  Controller1.pmOutfeeder1_goLayerCount -> SC_PM_PLC.pf2_GILayerCount
  Controller1.pmOutfeeder1_goProductCount -> SC_PM_PLC.pf2_GIProductCount
  Controller1.pmOutfeeder1_goProduct -> SC_PM_PLC.pf2_GOProductSignal
  Controller1.pmOutfeeder1_goFormat -> SC_PM_PLC.pf2_GOFormatSignal
  Controller1.pmOutfeeder1_doOpSetCompl -> SC_PM_PLC.pf2_DIOpSetCompl
  PalletDispenser 1300_1300_300.Shown_ToPick -> SC_PM_PLC.pf3_DIShown_ToPick
  SC_PM_PLC.pf3_DOClear_ToPick -> PalletDispenser 1300_1300_300.Clear_ToPick
  SC_PM_PLC.pf3_DOEnqueue_ToPick -> PalletDispenser 1300_1300_300.Enqueue_ToPick
  PalletDispenser 1300_1300_300.GO_ProdSel_ToPick -> SC_PM_PLC.pf3_GI_ProdSel_ToPick
  PalletDispenser 1300_1300_300.GO_FormSel_ToPick -> SC_PM_PLC.pf3_GI_FormSel_ToPick
  SC_PM_PLC.pf3_GO_ProdSel_ToPick -> PalletDispenser 1300_1300_300.GI_ProdSel_ToPick
  SC_PM_PLC.pf3_GO_FormSel_ToPick -> PalletDispenser 1300_1300_300.GI_FormSel_ToPick
  PalletDispenser 1300_1300_300.Clear_Placed_Finished -> SC_PM_PLC.pf3_DIClear_Placed_Finished
  SC_PM_PLC.pf3_DOClear_Placed -> PalletDispenser 1300_1300_300.Clear_Placed
  SC_PM_PLC.pf3_DOEnqueue_Placed -> PalletDispenser 1300_1300_300.Enqueue_Placed
  SC_PM_PLC.pf3_DOEnqueue_PlacedRequest -> PalletDispenser 1300_1300_300.Enqueue_IOPlacedRequest
  PalletDispenser 1300_1300_300.GO_ProdSel_PlacedRequest -> SC_PM_PLC.pf3_GI_ProdSel_PlacedRequest
  PalletDispenser 1300_1300_300.GO_FormSel_PlacedRequest -> SC_PM_PLC.pf3_GI_FormSel_PlacedRequest
  SC_PM_PLC.pf3_GO_ProdSel_PlacedRequest -> PalletDispenser 1300_1300_300.GI_ProdSel_PlacedRequest
  SC_PM_PLC.pf3_GO_FormSel_PlacedRequest -> PalletDispenser 1300_1300_300.GI_FormSel_PlacedRequest
  PalletDispenser 1300_1300_300.IsReady_IOPlacedRequest -> SC_PM_PLC.pf3_DIIsReady_IOPlacedRequest
  SC_PM_PLC.pf3_DOReset -> PalletDispenser 1300_1300_300.Reset
  Controller1.pmPallet1_doPosReqTrig -> SC_PM_PLC.pf3_DIPosReqTrig
  Controller1.pmPallet1_goLayerCount -> SC_PM_PLC.pf3_GILayerCount
  Controller1.pmPallet1_goProductCount -> SC_PM_PLC.pf3_GIProductCount
  Controller1.pmPallet1_goProduct -> SC_PM_PLC.pf3_GOProductSignal
  Controller1.pmPallet1_goFormat -> SC_PM_PLC.pf3_GOFormatSignal
  Controller1.pmPallet1_doOpSetCompl -> SC_PM_PLC.pf3_DIOpSetCompl
  FlexGripper 2.0_Vacuum_Pallet.ReleasedObject => SC_PM_PLC.con0_T_ROB1_ObjectReleased
  SC_PM_PLC.pf1_Product_ToPick => Conveyor_600.Product_ToPick
  SC_PM_PLC.pf1_PreparationTime_ToPick => Conveyor_600.PreparationTime_ToPick
  SC_PM_PLC.pf1_Product_Placed => Conveyor_600.Product_Placed
  SC_PM_PLC.pf1_ClearTime_Placed => Conveyor_600.ClearTime_Placed
  SC_PM_PLC.pf2_Product_ToPick => Outfeeder_1320.Product_ToPick
  SC_PM_PLC.pf2_PreparationTime_ToPick => Outfeeder_1320.PreparationTime_ToPick
  SC_PM_PLC.pf2_Product_Placed => Outfeeder_1320.Product_Placed
  SC_PM_PLC.pf2_ClearTime_Placed => Outfeeder_1320.ClearTime_Placed
  SC_PM_PLC.pf3_Product_ToPick => PalletDispenser 1300_1300_300.Product_ToPick
  SC_PM_PLC.pf3_PreparationTime_ToPick => PalletDispenser 1300_1300_300.PreparationTime_ToPick
  SC_PM_PLC.pf3_Product_Placed => PalletDispenser 1300_1300_300.Product_Placed
  SC_PM_PLC.pf3_ClearTime_Placed => PalletDispenser 1300_1300_300.ClearTime_Placed
Targets, tools, work objects and paths stored in the station, written as RAPID:
! task T_ROB1
MODULE pmrcUser
  TASK PERS wobjdata pmInfeeder1_WObj:=[FALSE,TRUE,"",[[200,2100,270],[0.707106781,0,0,0.707106781]],[[0,0,0],[1,0,0,0]]];
  TASK PERS wobjdata pmInfeeder2_WObj:=[FALSE,TRUE,"",[[0,0,-500],[1,0,0,0]],[[0,0,0],[1,0,0,0]]];
  TASK PERS wobjdata pmInfeeder3_WObj:=[FALSE,TRUE,"",[[0,0,-500],[1,0,0,0]],[[0,0,0],[1,0,0,0]]];
  TASK PERS wobjdata pmInfeeder4_WObj:=[FALSE,TRUE,"",[[0,0,-500],[1,0,0,0]],[[0,0,0],[1,0,0,0]]];
  TASK PERS wobjdata pmOutfeeder1_WObj:=[FALSE,TRUE,"",[[1660,580,-80.253967285],[1,0,0,0]],[[0,0,0],[1,0,0,0]]];
  TASK PERS wobjdata pmOutfeeder2_WObj:=[FALSE,TRUE,"",[[0,0,-500],[1,0,0,0]],[[0,0,0],[1,0,0,0]]];
  TASK PERS wobjdata pmOutfeeder3_WObj:=[FALSE,TRUE,"",[[0,0,-500],[1,0,0,0]],[[0,0,0],[1,0,0,0]]];
  TASK PERS wobjdata pmOutfeeder4_WObj:=[FALSE,TRUE,"",[[0,0,-500],[1,0,0,0]],[[0,0,0],[1,0,0,0]]];
  TASK PERS wobjdata pmPallet1_WObj:=[FALSE,TRUE,"",[[934.960859983,-1595.677464876,-292],[0.707106781,0,0,-0.707106781]],[[0,0,0],[1,0,0,0]]];
  TASK PERS wobjdata pmSlipsheet1_WObj:=[FALSE,TRUE,"",[[0,0,-500],[1,0,0,0]],[[0,0,0],[1,0,0,0]]];
  TASK PERS tooldata pmPickTool1:=[TRUE,[[0,0,0],[1,0,0,0]],[1,[0,0,10],[1,0,0,0],0.01,0.01,0.01]];
  TASK PERS tooldata pmSearchTool1:=[TRUE,[[0,0,0],[1,0,0,0]],[1,[0,0,10],[1,0,0,0],0.01,0.01,0.01]];
  TASK PERS tooldata tVacuum:=[TRUE,[[0.12,0.029,163.808],[0.99999998,0,0,-0.000200713]],[95,[0,0,10],[1,0,0,0],0.158,0.158,0.158]];
  TASK PERS tooldata tPalletPicker:=[TRUE,[[0.12,0.029,230.105],[0.99999998,0,0,-0.000200713]],[95,[0,0,10],[1,0,0,0],0.158,0.158,0.158]];
ENDMODULE

! task T_ROB1
MODULE pmrcSys
  TASK PERS wobjdata pm_home_WObj:=[FALSE,TRUE,"",[[0,0,-500],[1,0,0,0]],[[0,0,0],[1,0,0,0]]];
ENDMODULE

